Fanuc KAREL source: kd00006.KL

-- PROVISIONAL review KL for V1013-1; original PC SHA256 76a51bc8b8f342e50625efd9a5ecfec9bbb8d3f9e668e241f1259b6b32d6daa4
-- Incomplete behavior may be omitted. Consult companion uncertainty JSON. Do not deploy.
PROGRAM KD00006
%NOLOCKGROUP
VAR
  I : INTEGER
  J : INTEGER
  B : BOOLEAN
  R : REAL
  S : STRING[80]
BEGIN
  -- UNRESOLVED_PC offsets 5-12; opcodes 9D,23
  -- UNRESOLVED_PC offsets 17-21; opcodes 7F
END KD00006
